// TIA Portal V20 export
FUNCTION "CollectAlarms" : Void   // FC96, LAD
TITLE = Alarm Collector Unit
// Collects alarms from the respective level and categorises the alarms into the different alarm classes.
// stored: Namespace Unit1.Em5, SetENOAutomatically false
   VAR_INPUT
      resetAlarms : Bool;
      disableAlarms : Bool;
   END_VAR
   VAR_OUTPUT
      commandsToUnit : "LUC_typeStateCommands";   // Feedback to the unit
   END_VAR
   VAR CONSTANT
      DelayTime : Time := T#300ms;
      TRUE : Bool := TRUE;
      FALSE : Bool := FALSE;
   END_VAR
BEGIN

REGION Network 1: Reset Alarms
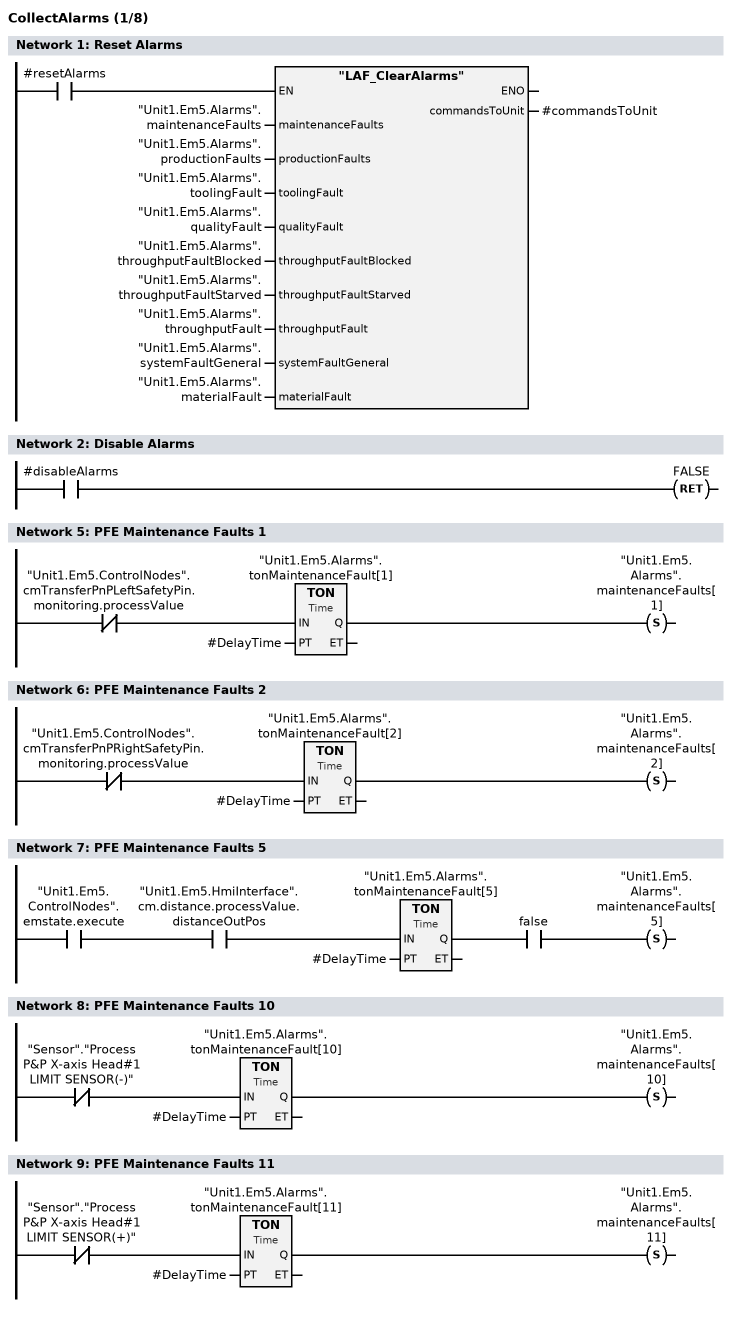
   RUNG wire#powerrail
      Contact( #resetAlarms )
      "LAF_ClearAlarms"(maintenanceFaults := "Unit1.Em5.Alarms".maintenanceFaults, productionFaults := "Unit1.Em5.Alarms".productionFaults, toolingFault := "Unit1.Em5.Alarms".toolingFault, qualityFault := "Unit1.Em5.Alarms".qualityFault, throughputFaultBlocked := "Unit1.Em5.Alarms".throughputFaultBlocked, throughputFaultStarved := "Unit1.Em5.Alarms".throughputFaultStarved, throughputFault := "Unit1.Em5.Alarms".throughputFault, systemFaultGeneral := "Unit1.Em5.Alarms".systemFaultGeneral, materialFault := "Unit1.Em5.Alarms".materialFault, commandsToUnit => #commandsToUnit)
   END_RUNG
   // the same network as SCL:
   IF #resetAlarms THEN
       "LAF_ClearAlarms"(maintenanceFaults := "Unit1.Em5.Alarms".maintenanceFaults,
                         productionFaults := "Unit1.Em5.Alarms".productionFaults,
                         toolingFault := "Unit1.Em5.Alarms".toolingFault,
                         qualityFault := "Unit1.Em5.Alarms".qualityFault,
                         throughputFaultBlocked := "Unit1.Em5.Alarms".throughputFaultBlocked,
                         throughputFaultStarved := "Unit1.Em5.Alarms".throughputFaultStarved,
                         throughputFault := "Unit1.Em5.Alarms".throughputFault,
                         systemFaultGeneral := "Unit1.Em5.Alarms".systemFaultGeneral,
                         materialFault := "Unit1.Em5.Alarms".materialFault,
                         commandsToUnit => #commandsToUnit);
   END_IF;
END_REGION

REGION Network 2: Disable Alarms
   RUNG wire#powerrail
      Contact( #disableAlarms )
      ReturnCoil( FALSE )
   END_RUNG
   // the same network as SCL:
   IF #disableAlarms THEN
       ENO := FALSE;
       RETURN;
   END_IF;
END_REGION

REGION Network 3: *************** Fault ************************
END_REGION

REGION Network 4: PFE Maintenance Faults 0
END_REGION

REGION Network 5: PFE Maintenance Faults 1
   RUNG wire#powerrail
      I_Contact( "Unit1.Em5.ControlNodes".cmTransferPnPLeftSafetyPin.monitoring.processValue )
      { S7_Templates := "time_type := Time" } "Unit1.Em5.Alarms".tonMaintenanceFault[1].TON(pt := #DelayTime, et =>)
      S_Coil( "Unit1.Em5.Alarms".maintenanceFaults[1] )
   END_RUNG
   // the same network as SCL:
   "Unit1.Em5.Alarms".tonMaintenanceFault[1].TON(IN := NOT "Unit1.Em5.ControlNodes".cmTransferPnPLeftSafetyPin.monitoring.processValue,
                           PT := #DelayTime);
   IF "Unit1.Em5.Alarms".tonMaintenanceFault[1].Q THEN
       "Unit1.Em5.Alarms".maintenanceFaults[1] := TRUE;
   END_IF;
END_REGION

REGION Network 6: PFE Maintenance Faults 2
   RUNG wire#powerrail
      I_Contact( "Unit1.Em5.ControlNodes".cmTransferPnPRightSafetyPin.monitoring.processValue )
      { S7_Templates := "time_type := Time" } "Unit1.Em5.Alarms".tonMaintenanceFault[2].TON(pt := #DelayTime, et =>)
      S_Coil( "Unit1.Em5.Alarms".maintenanceFaults[2] )
   END_RUNG
   // the same network as SCL:
   "Unit1.Em5.Alarms".tonMaintenanceFault[2].TON(IN := NOT "Unit1.Em5.ControlNodes".cmTransferPnPRightSafetyPin.monitoring.processValue,
                           PT := #DelayTime);
   IF "Unit1.Em5.Alarms".tonMaintenanceFault[2].Q THEN
       "Unit1.Em5.Alarms".maintenanceFaults[2] := TRUE;
   END_IF;
END_REGION

REGION Network 7: PFE Maintenance Faults 5
   RUNG wire#powerrail
      Contact( "Unit1.Em5.ControlNodes".emstate.execute )
      Contact( "Unit1.Em5.HmiInterface".cm.distance.processValue.distanceOutPos )
      { S7_Templates := "time_type := Time" } "Unit1.Em5.Alarms".tonMaintenanceFault[5].TON(pt := #DelayTime, et =>)
      Contact( false )
      S_Coil( "Unit1.Em5.Alarms".maintenanceFaults[5] )
   END_RUNG
   // the same network as SCL:
   "Unit1.Em5.Alarms".tonMaintenanceFault[5].TON(IN := "Unit1.Em5.ControlNodes".emstate.execute AND "Unit1.Em5.HmiInterface".cm.distance.processValue.distanceOutPos,
                           PT := #DelayTime);
   IF "Unit1.Em5.Alarms".tonMaintenanceFault[5].Q AND false THEN
       "Unit1.Em5.Alarms".maintenanceFaults[5] := TRUE;
   END_IF;
END_REGION

REGION Network 8: PFE Maintenance Faults 10
   RUNG wire#powerrail
      I_Contact( "Sensor"."Process P&P X-axis Head#1 LIMIT SENSOR(-)" )
      { S7_Templates := "time_type := Time" } "Unit1.Em5.Alarms".tonMaintenanceFault[10].TON(pt := #DelayTime, et =>)
      S_Coil( "Unit1.Em5.Alarms".maintenanceFaults[10] )
   END_RUNG
   // the same network as SCL:
   "Unit1.Em5.Alarms".tonMaintenanceFault[10].TON(IN := NOT "Sensor"."Process P&P X-axis Head#1 LIMIT SENSOR(-)",
                           PT := #DelayTime);
   IF "Unit1.Em5.Alarms".tonMaintenanceFault[10].Q THEN
       "Unit1.Em5.Alarms".maintenanceFaults[10] := TRUE;
   END_IF;
END_REGION

REGION Network 9: PFE Maintenance Faults 11
   RUNG wire#powerrail
      I_Contact( "Sensor"."Process P&P X-axis Head#1 LIMIT SENSOR(+)" )
      { S7_Templates := "time_type := Time" } "Unit1.Em5.Alarms".tonMaintenanceFault[11].TON(pt := #DelayTime, et =>)
      S_Coil( "Unit1.Em5.Alarms".maintenanceFaults[11] )
   END_RUNG
   // the same network as SCL:
   "Unit1.Em5.Alarms".tonMaintenanceFault[11].TON(IN := NOT "Sensor"."Process P&P X-axis Head#1 LIMIT SENSOR(+)",
                           PT := #DelayTime);
   IF "Unit1.Em5.Alarms".tonMaintenanceFault[11].Q THEN
       "Unit1.Em5.Alarms".maintenanceFaults[11] := TRUE;
   END_IF;
END_REGION

REGION Network 10: PFE Maintenance Faults 12
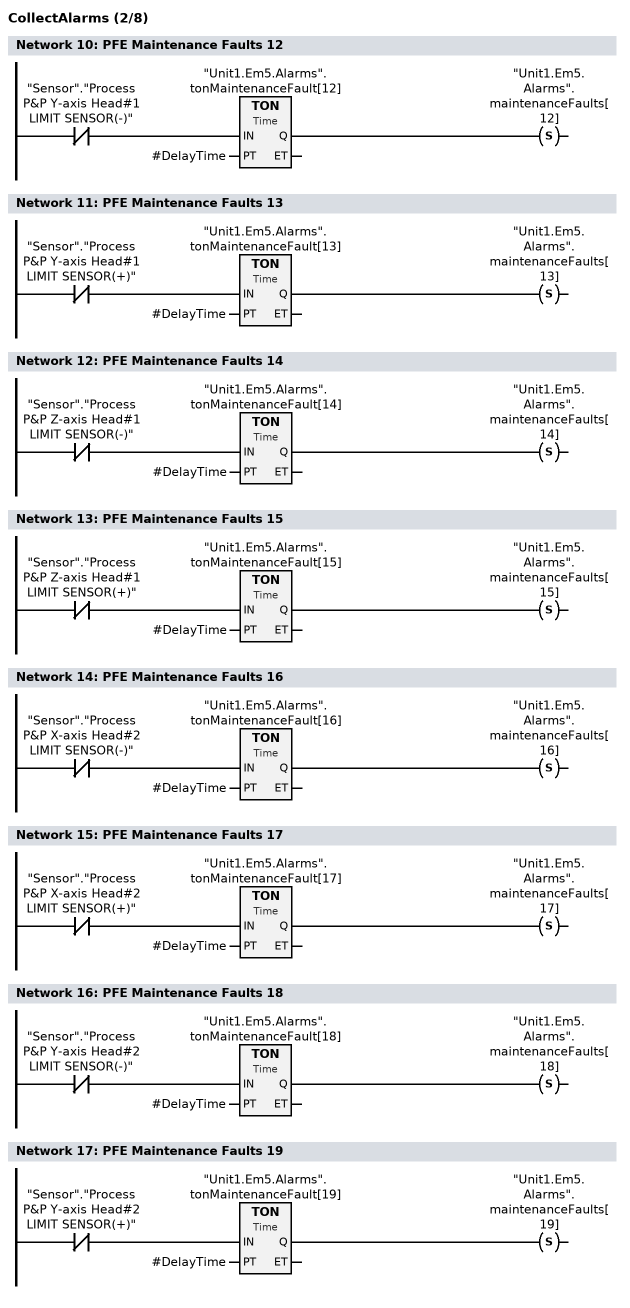
   RUNG wire#powerrail
      I_Contact( "Sensor"."Process P&P Y-axis Head#1 LIMIT SENSOR(-)" )
      { S7_Templates := "time_type := Time" } "Unit1.Em5.Alarms".tonMaintenanceFault[12].TON(pt := #DelayTime, et =>)
      S_Coil( "Unit1.Em5.Alarms".maintenanceFaults[12] )
   END_RUNG
   // the same network as SCL:
   "Unit1.Em5.Alarms".tonMaintenanceFault[12].TON(IN := NOT "Sensor"."Process P&P Y-axis Head#1 LIMIT SENSOR(-)",
                           PT := #DelayTime);
   IF "Unit1.Em5.Alarms".tonMaintenanceFault[12].Q THEN
       "Unit1.Em5.Alarms".maintenanceFaults[12] := TRUE;
   END_IF;
END_REGION

REGION Network 11: PFE Maintenance Faults 13
   RUNG wire#powerrail
      I_Contact( "Sensor"."Process P&P Y-axis Head#1 LIMIT SENSOR(+)" )
      { S7_Templates := "time_type := Time" } "Unit1.Em5.Alarms".tonMaintenanceFault[13].TON(pt := #DelayTime, et =>)
      S_Coil( "Unit1.Em5.Alarms".maintenanceFaults[13] )
   END_RUNG
   // the same network as SCL:
   "Unit1.Em5.Alarms".tonMaintenanceFault[13].TON(IN := NOT "Sensor"."Process P&P Y-axis Head#1 LIMIT SENSOR(+)",
                           PT := #DelayTime);
   IF "Unit1.Em5.Alarms".tonMaintenanceFault[13].Q THEN
       "Unit1.Em5.Alarms".maintenanceFaults[13] := TRUE;
   END_IF;
END_REGION

REGION Network 12: PFE Maintenance Faults 14
   RUNG wire#powerrail
      I_Contact( "Sensor"."Process P&P Z-axis Head#1 LIMIT SENSOR(-)" )
      { S7_Templates := "time_type := Time" } "Unit1.Em5.Alarms".tonMaintenanceFault[14].TON(pt := #DelayTime, et =>)
      S_Coil( "Unit1.Em5.Alarms".maintenanceFaults[14] )
   END_RUNG
   // the same network as SCL:
   "Unit1.Em5.Alarms".tonMaintenanceFault[14].TON(IN := NOT "Sensor"."Process P&P Z-axis Head#1 LIMIT SENSOR(-)",
                           PT := #DelayTime);
   IF "Unit1.Em5.Alarms".tonMaintenanceFault[14].Q THEN
       "Unit1.Em5.Alarms".maintenanceFaults[14] := TRUE;
   END_IF;
END_REGION

REGION Network 13: PFE Maintenance Faults 15
   RUNG wire#powerrail
      I_Contact( "Sensor"."Process P&P Z-axis Head#1 LIMIT SENSOR(+)" )
      { S7_Templates := "time_type := Time" } "Unit1.Em5.Alarms".tonMaintenanceFault[15].TON(pt := #DelayTime, et =>)
      S_Coil( "Unit1.Em5.Alarms".maintenanceFaults[15] )
   END_RUNG
   // the same network as SCL:
   "Unit1.Em5.Alarms".tonMaintenanceFault[15].TON(IN := NOT "Sensor"."Process P&P Z-axis Head#1 LIMIT SENSOR(+)",
                           PT := #DelayTime);
   IF "Unit1.Em5.Alarms".tonMaintenanceFault[15].Q THEN
       "Unit1.Em5.Alarms".maintenanceFaults[15] := TRUE;
   END_IF;
END_REGION

REGION Network 14: PFE Maintenance Faults 16
   RUNG wire#powerrail
      I_Contact( "Sensor"."Process P&P X-axis Head#2 LIMIT SENSOR(-)" )
      { S7_Templates := "time_type := Time" } "Unit1.Em5.Alarms".tonMaintenanceFault[16].TON(pt := #DelayTime, et =>)
      S_Coil( "Unit1.Em5.Alarms".maintenanceFaults[16] )
   END_RUNG
   // the same network as SCL:
   "Unit1.Em5.Alarms".tonMaintenanceFault[16].TON(IN := NOT "Sensor"."Process P&P X-axis Head#2 LIMIT SENSOR(-)",
                           PT := #DelayTime);
   IF "Unit1.Em5.Alarms".tonMaintenanceFault[16].Q THEN
       "Unit1.Em5.Alarms".maintenanceFaults[16] := TRUE;
   END_IF;
END_REGION

REGION Network 15: PFE Maintenance Faults 17
   RUNG wire#powerrail
      I_Contact( "Sensor"."Process P&P X-axis Head#2 LIMIT SENSOR(+)" )
      { S7_Templates := "time_type := Time" } "Unit1.Em5.Alarms".tonMaintenanceFault[17].TON(pt := #DelayTime, et =>)
      S_Coil( "Unit1.Em5.Alarms".maintenanceFaults[17] )
   END_RUNG
   // the same network as SCL:
   "Unit1.Em5.Alarms".tonMaintenanceFault[17].TON(IN := NOT "Sensor"."Process P&P X-axis Head#2 LIMIT SENSOR(+)",
                           PT := #DelayTime);
   IF "Unit1.Em5.Alarms".tonMaintenanceFault[17].Q THEN
       "Unit1.Em5.Alarms".maintenanceFaults[17] := TRUE;
   END_IF;
END_REGION

REGION Network 16: PFE Maintenance Faults 18
   RUNG wire#powerrail
      I_Contact( "Sensor"."Process P&P Y-axis Head#2 LIMIT SENSOR(-)" )
      { S7_Templates := "time_type := Time" } "Unit1.Em5.Alarms".tonMaintenanceFault[18].TON(pt := #DelayTime, et =>)
      S_Coil( "Unit1.Em5.Alarms".maintenanceFaults[18] )
   END_RUNG
   // the same network as SCL:
   "Unit1.Em5.Alarms".tonMaintenanceFault[18].TON(IN := NOT "Sensor"."Process P&P Y-axis Head#2 LIMIT SENSOR(-)",
                           PT := #DelayTime);
   IF "Unit1.Em5.Alarms".tonMaintenanceFault[18].Q THEN
       "Unit1.Em5.Alarms".maintenanceFaults[18] := TRUE;
   END_IF;
END_REGION

REGION Network 17: PFE Maintenance Faults 19
   RUNG wire#powerrail
      I_Contact( "Sensor"."Process P&P Y-axis Head#2 LIMIT SENSOR(+)" )
      { S7_Templates := "time_type := Time" } "Unit1.Em5.Alarms".tonMaintenanceFault[19].TON(pt := #DelayTime, et =>)
      S_Coil( "Unit1.Em5.Alarms".maintenanceFaults[19] )
   END_RUNG
   // the same network as SCL:
   "Unit1.Em5.Alarms".tonMaintenanceFault[19].TON(IN := NOT "Sensor"."Process P&P Y-axis Head#2 LIMIT SENSOR(+)",
                           PT := #DelayTime);
   IF "Unit1.Em5.Alarms".tonMaintenanceFault[19].Q THEN
       "Unit1.Em5.Alarms".maintenanceFaults[19] := TRUE;
   END_IF;
END_REGION

REGION Network 18: PFE Maintenance Faults 20
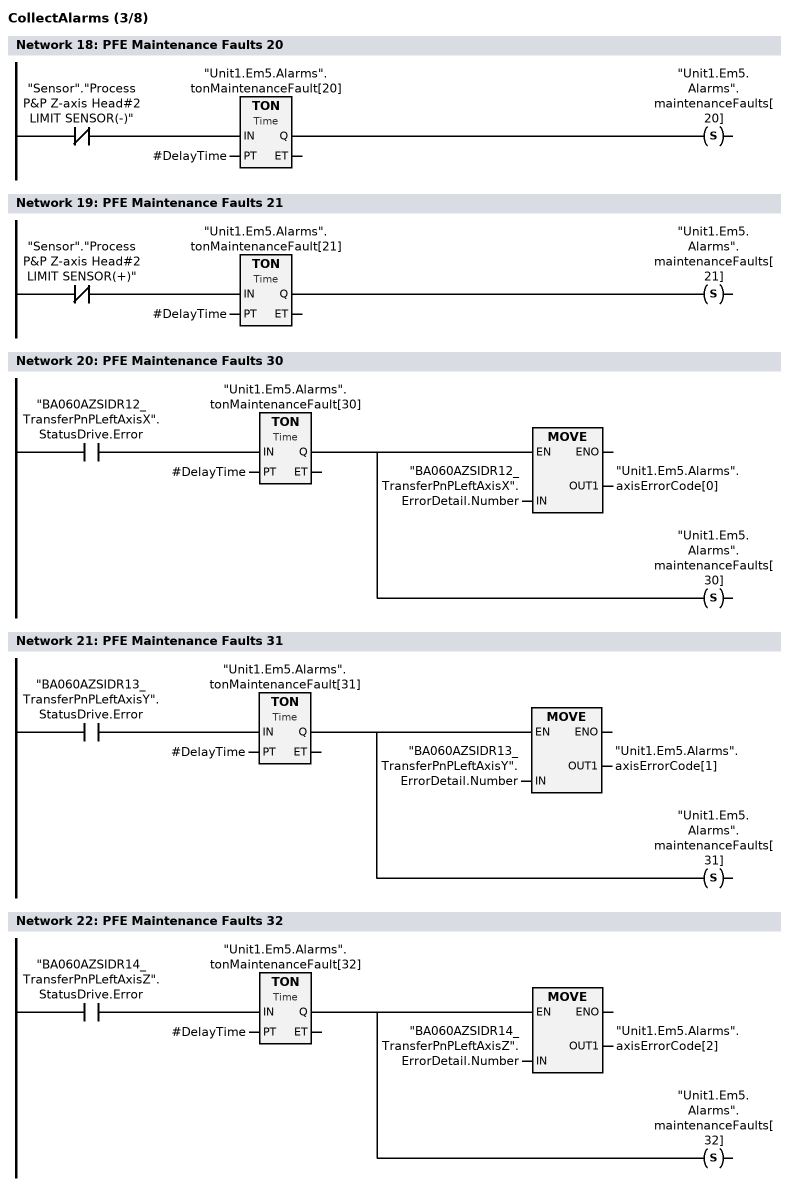
   RUNG wire#powerrail
      I_Contact( "Sensor"."Process P&P Z-axis Head#2 LIMIT SENSOR(-)" )
      { S7_Templates := "time_type := Time" } "Unit1.Em5.Alarms".tonMaintenanceFault[20].TON(pt := #DelayTime, et =>)
      S_Coil( "Unit1.Em5.Alarms".maintenanceFaults[20] )
   END_RUNG
   // the same network as SCL:
   "Unit1.Em5.Alarms".tonMaintenanceFault[20].TON(IN := NOT "Sensor"."Process P&P Z-axis Head#2 LIMIT SENSOR(-)",
                           PT := #DelayTime);
   IF "Unit1.Em5.Alarms".tonMaintenanceFault[20].Q THEN
       "Unit1.Em5.Alarms".maintenanceFaults[20] := TRUE;
   END_IF;
END_REGION

REGION Network 19: PFE Maintenance Faults 21
   RUNG wire#powerrail
      I_Contact( "Sensor"."Process P&P Z-axis Head#2 LIMIT SENSOR(+)" )
      { S7_Templates := "time_type := Time" } "Unit1.Em5.Alarms".tonMaintenanceFault[21].TON(pt := #DelayTime, et =>)
      S_Coil( "Unit1.Em5.Alarms".maintenanceFaults[21] )
   END_RUNG
   // the same network as SCL:
   "Unit1.Em5.Alarms".tonMaintenanceFault[21].TON(IN := NOT "Sensor"."Process P&P Z-axis Head#2 LIMIT SENSOR(+)",
                           PT := #DelayTime);
   IF "Unit1.Em5.Alarms".tonMaintenanceFault[21].Q THEN
       "Unit1.Em5.Alarms".maintenanceFaults[21] := TRUE;
   END_IF;
END_REGION

REGION Network 20: PFE Maintenance Faults 30
   RUNG wire#powerrail
      Contact( "BA060AZSIDR12_TransferPnPLeftAxisX".StatusDrive.Error )
      { S7_Templates := "time_type := Time" } "Unit1.Em5.Alarms".tonMaintenanceFault[30].TON(pt := #DelayTime, et =>)
      wire#w1
      Move(in := "BA060AZSIDR12_TransferPnPLeftAxisX".ErrorDetail.Number, out1 => "Unit1.Em5.Alarms".axisErrorCode[0])
   END_RUNG
   RUNG wire#w1
      S_Coil( "Unit1.Em5.Alarms".maintenanceFaults[30] )
   END_RUNG
   // the same network as SCL:
   "Unit1.Em5.Alarms".tonMaintenanceFault[30].TON(IN := "BA060AZSIDR12_TransferPnPLeftAxisX".StatusDrive.Error,
                           PT := #DelayTime);
   IF "Unit1.Em5.Alarms".tonMaintenanceFault[30].Q THEN
       "Unit1.Em5.Alarms".axisErrorCode[0] := "BA060AZSIDR12_TransferPnPLeftAxisX".ErrorDetail.Number;
       "Unit1.Em5.Alarms".maintenanceFaults[30] := TRUE;
   END_IF;
END_REGION

REGION Network 21: PFE Maintenance Faults 31
   RUNG wire#powerrail
      Contact( "BA060AZSIDR13_TransferPnPLeftAxisY".StatusDrive.Error )
      { S7_Templates := "time_type := Time" } "Unit1.Em5.Alarms".tonMaintenanceFault[31].TON(pt := #DelayTime, et =>)
      wire#w1
      Move(in := "BA060AZSIDR13_TransferPnPLeftAxisY".ErrorDetail.Number, out1 => "Unit1.Em5.Alarms".axisErrorCode[1])
   END_RUNG
   RUNG wire#w1
      S_Coil( "Unit1.Em5.Alarms".maintenanceFaults[31] )
   END_RUNG
   // the same network as SCL:
   "Unit1.Em5.Alarms".tonMaintenanceFault[31].TON(IN := "BA060AZSIDR13_TransferPnPLeftAxisY".StatusDrive.Error,
                           PT := #DelayTime);
   IF "Unit1.Em5.Alarms".tonMaintenanceFault[31].Q THEN
       "Unit1.Em5.Alarms".axisErrorCode[1] := "BA060AZSIDR13_TransferPnPLeftAxisY".ErrorDetail.Number;
       "Unit1.Em5.Alarms".maintenanceFaults[31] := TRUE;
   END_IF;
END_REGION

REGION Network 22: PFE Maintenance Faults 32
   RUNG wire#powerrail
      Contact( "BA060AZSIDR14_TransferPnPLeftAxisZ".StatusDrive.Error )
      { S7_Templates := "time_type := Time" } "Unit1.Em5.Alarms".tonMaintenanceFault[32].TON(pt := #DelayTime, et =>)
      wire#w1
      Move(in := "BA060AZSIDR14_TransferPnPLeftAxisZ".ErrorDetail.Number, out1 => "Unit1.Em5.Alarms".axisErrorCode[2])
   END_RUNG
   RUNG wire#w1
      S_Coil( "Unit1.Em5.Alarms".maintenanceFaults[32] )
   END_RUNG
   // the same network as SCL:
   "Unit1.Em5.Alarms".tonMaintenanceFault[32].TON(IN := "BA060AZSIDR14_TransferPnPLeftAxisZ".StatusDrive.Error,
                           PT := #DelayTime);
   IF "Unit1.Em5.Alarms".tonMaintenanceFault[32].Q THEN
       "Unit1.Em5.Alarms".axisErrorCode[2] := "BA060AZSIDR14_TransferPnPLeftAxisZ".ErrorDetail.Number;
       "Unit1.Em5.Alarms".maintenanceFaults[32] := TRUE;
   END_IF;
END_REGION

REGION Network 23: PFE Maintenance Faults 33
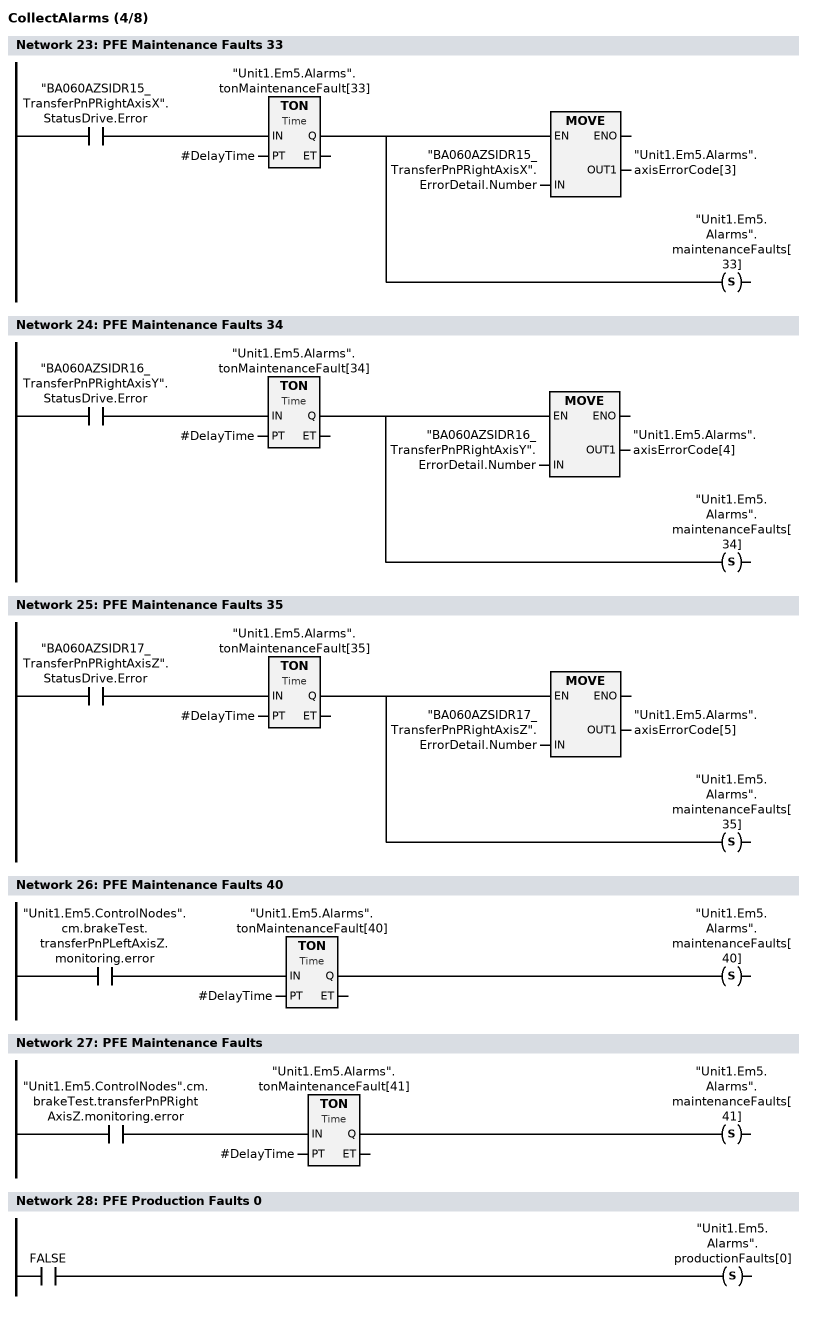
   RUNG wire#powerrail
      Contact( "BA060AZSIDR15_TransferPnPRightAxisX".StatusDrive.Error )
      { S7_Templates := "time_type := Time" } "Unit1.Em5.Alarms".tonMaintenanceFault[33].TON(pt := #DelayTime, et =>)
      wire#w1
      Move(in := "BA060AZSIDR15_TransferPnPRightAxisX".ErrorDetail.Number, out1 => "Unit1.Em5.Alarms".axisErrorCode[3])
   END_RUNG
   RUNG wire#w1
      S_Coil( "Unit1.Em5.Alarms".maintenanceFaults[33] )
   END_RUNG
   // the same network as SCL:
   "Unit1.Em5.Alarms".tonMaintenanceFault[33].TON(IN := "BA060AZSIDR15_TransferPnPRightAxisX".StatusDrive.Error,
                           PT := #DelayTime);
   IF "Unit1.Em5.Alarms".tonMaintenanceFault[33].Q THEN
       "Unit1.Em5.Alarms".axisErrorCode[3] := "BA060AZSIDR15_TransferPnPRightAxisX".ErrorDetail.Number;
       "Unit1.Em5.Alarms".maintenanceFaults[33] := TRUE;
   END_IF;
END_REGION

REGION Network 24: PFE Maintenance Faults 34
   RUNG wire#powerrail
      Contact( "BA060AZSIDR16_TransferPnPRightAxisY".StatusDrive.Error )
      { S7_Templates := "time_type := Time" } "Unit1.Em5.Alarms".tonMaintenanceFault[34].TON(pt := #DelayTime, et =>)
      wire#w1
      Move(in := "BA060AZSIDR16_TransferPnPRightAxisY".ErrorDetail.Number, out1 => "Unit1.Em5.Alarms".axisErrorCode[4])
   END_RUNG
   RUNG wire#w1
      S_Coil( "Unit1.Em5.Alarms".maintenanceFaults[34] )
   END_RUNG
   // the same network as SCL:
   "Unit1.Em5.Alarms".tonMaintenanceFault[34].TON(IN := "BA060AZSIDR16_TransferPnPRightAxisY".StatusDrive.Error,
                           PT := #DelayTime);
   IF "Unit1.Em5.Alarms".tonMaintenanceFault[34].Q THEN
       "Unit1.Em5.Alarms".axisErrorCode[4] := "BA060AZSIDR16_TransferPnPRightAxisY".ErrorDetail.Number;
       "Unit1.Em5.Alarms".maintenanceFaults[34] := TRUE;
   END_IF;
END_REGION

REGION Network 25: PFE Maintenance Faults 35
   RUNG wire#powerrail
      Contact( "BA060AZSIDR17_TransferPnPRightAxisZ".StatusDrive.Error )
      { S7_Templates := "time_type := Time" } "Unit1.Em5.Alarms".tonMaintenanceFault[35].TON(pt := #DelayTime, et =>)
      wire#w1
      Move(in := "BA060AZSIDR17_TransferPnPRightAxisZ".ErrorDetail.Number, out1 => "Unit1.Em5.Alarms".axisErrorCode[5])
   END_RUNG
   RUNG wire#w1
      S_Coil( "Unit1.Em5.Alarms".maintenanceFaults[35] )
   END_RUNG
   // the same network as SCL:
   "Unit1.Em5.Alarms".tonMaintenanceFault[35].TON(IN := "BA060AZSIDR17_TransferPnPRightAxisZ".StatusDrive.Error,
                           PT := #DelayTime);
   IF "Unit1.Em5.Alarms".tonMaintenanceFault[35].Q THEN
       "Unit1.Em5.Alarms".axisErrorCode[5] := "BA060AZSIDR17_TransferPnPRightAxisZ".ErrorDetail.Number;
       "Unit1.Em5.Alarms".maintenanceFaults[35] := TRUE;
   END_IF;
END_REGION

REGION Network 26: PFE Maintenance Faults 40
   RUNG wire#powerrail
      Contact( "Unit1.Em5.ControlNodes".cm.brakeTest.transferPnPLeftAxisZ.monitoring.error )
      { S7_Templates := "time_type := Time" } "Unit1.Em5.Alarms".tonMaintenanceFault[40].TON(pt := #DelayTime, et =>)
      S_Coil( "Unit1.Em5.Alarms".maintenanceFaults[40] )
   END_RUNG
   // the same network as SCL:
   "Unit1.Em5.Alarms".tonMaintenanceFault[40].TON(IN := "Unit1.Em5.ControlNodes".cm.brakeTest.transferPnPLeftAxisZ.monitoring.error,
                           PT := #DelayTime);
   IF "Unit1.Em5.Alarms".tonMaintenanceFault[40].Q THEN
       "Unit1.Em5.Alarms".maintenanceFaults[40] := TRUE;
   END_IF;
END_REGION

REGION Network 27: PFE Maintenance Faults
   RUNG wire#powerrail
      Contact( "Unit1.Em5.ControlNodes".cm.brakeTest.transferPnPRightAxisZ.monitoring.error )
      { S7_Templates := "time_type := Time" } "Unit1.Em5.Alarms".tonMaintenanceFault[41].TON(pt := #DelayTime, et =>)
      S_Coil( "Unit1.Em5.Alarms".maintenanceFaults[41] )
   END_RUNG
   // the same network as SCL:
   "Unit1.Em5.Alarms".tonMaintenanceFault[41].TON(IN := "Unit1.Em5.ControlNodes".cm.brakeTest.transferPnPRightAxisZ.monitoring.error,
                           PT := #DelayTime);
   IF "Unit1.Em5.Alarms".tonMaintenanceFault[41].Q THEN
       "Unit1.Em5.Alarms".maintenanceFaults[41] := TRUE;
   END_IF;
END_REGION

REGION Network 28: PFE Production Faults 0
   RUNG wire#powerrail
      Contact( FALSE )
      S_Coil( "Unit1.Em5.Alarms".productionFaults[0] )
   END_RUNG
   // the same network as SCL:
   IF FALSE THEN "Unit1.Em5.Alarms".productionFaults[0] := TRUE; END_IF;
END_REGION

REGION Network 29: PFE Production Faults 1
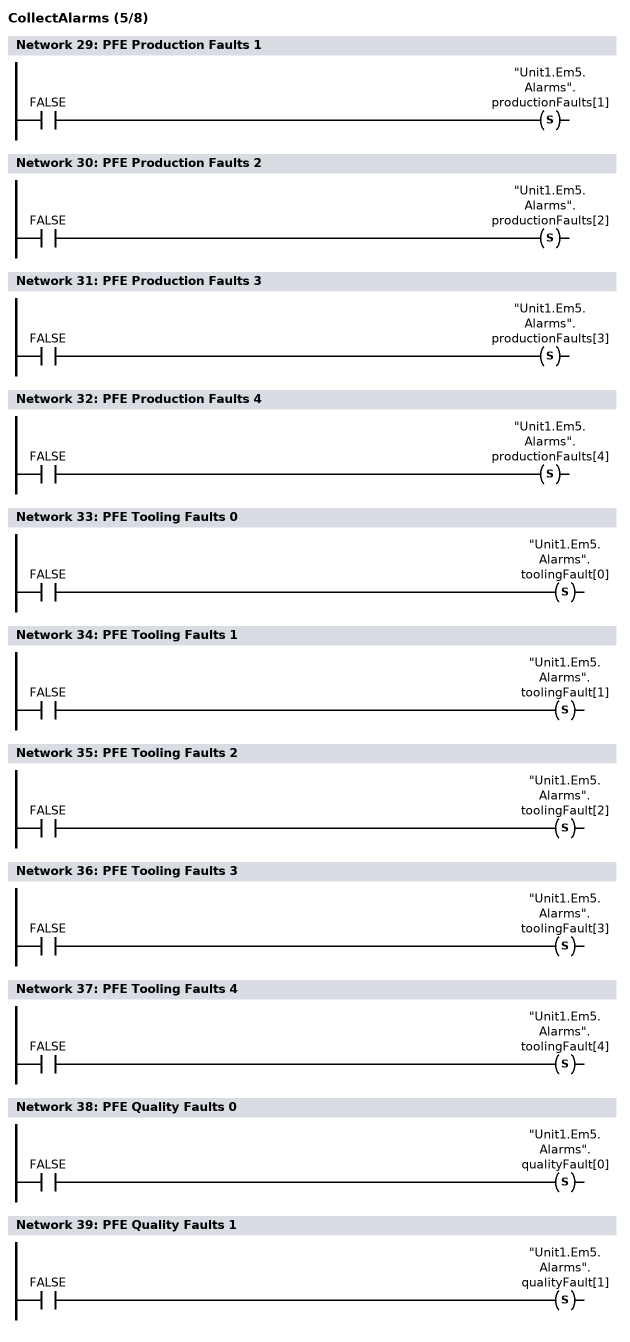
   RUNG wire#powerrail
      Contact( FALSE )
      S_Coil( "Unit1.Em5.Alarms".productionFaults[1] )
   END_RUNG
   // the same network as SCL:
   IF FALSE THEN "Unit1.Em5.Alarms".productionFaults[1] := TRUE; END_IF;
END_REGION

REGION Network 30: PFE Production Faults 2
   RUNG wire#powerrail
      Contact( FALSE )
      S_Coil( "Unit1.Em5.Alarms".productionFaults[2] )
   END_RUNG
   // the same network as SCL:
   IF FALSE THEN "Unit1.Em5.Alarms".productionFaults[2] := TRUE; END_IF;
END_REGION

REGION Network 31: PFE Production Faults 3
   RUNG wire#powerrail
      Contact( FALSE )
      S_Coil( "Unit1.Em5.Alarms".productionFaults[3] )
   END_RUNG
   // the same network as SCL:
   IF FALSE THEN "Unit1.Em5.Alarms".productionFaults[3] := TRUE; END_IF;
END_REGION

REGION Network 32: PFE Production Faults 4
   RUNG wire#powerrail
      Contact( FALSE )
      S_Coil( "Unit1.Em5.Alarms".productionFaults[4] )
   END_RUNG
   // the same network as SCL:
   IF FALSE THEN "Unit1.Em5.Alarms".productionFaults[4] := TRUE; END_IF;
END_REGION

REGION Network 33: PFE Tooling Faults 0
   RUNG wire#powerrail
      Contact( FALSE )
      S_Coil( "Unit1.Em5.Alarms".toolingFault[0] )
   END_RUNG
   // the same network as SCL:
   IF FALSE THEN "Unit1.Em5.Alarms".toolingFault[0] := TRUE; END_IF;
END_REGION

REGION Network 34: PFE Tooling Faults 1
   RUNG wire#powerrail
      Contact( FALSE )
      S_Coil( "Unit1.Em5.Alarms".toolingFault[1] )
   END_RUNG
   // the same network as SCL:
   IF FALSE THEN "Unit1.Em5.Alarms".toolingFault[1] := TRUE; END_IF;
END_REGION

REGION Network 35: PFE Tooling Faults 2
   RUNG wire#powerrail
      Contact( FALSE )
      S_Coil( "Unit1.Em5.Alarms".toolingFault[2] )
   END_RUNG
   // the same network as SCL:
   IF FALSE THEN "Unit1.Em5.Alarms".toolingFault[2] := TRUE; END_IF;
END_REGION

REGION Network 36: PFE Tooling Faults 3
   RUNG wire#powerrail
      Contact( FALSE )
      S_Coil( "Unit1.Em5.Alarms".toolingFault[3] )
   END_RUNG
   // the same network as SCL:
   IF FALSE THEN "Unit1.Em5.Alarms".toolingFault[3] := TRUE; END_IF;
END_REGION

REGION Network 37: PFE Tooling Faults 4
   RUNG wire#powerrail
      Contact( FALSE )
      S_Coil( "Unit1.Em5.Alarms".toolingFault[4] )
   END_RUNG
   // the same network as SCL:
   IF FALSE THEN "Unit1.Em5.Alarms".toolingFault[4] := TRUE; END_IF;
END_REGION

REGION Network 38: PFE Quality Faults 0
   RUNG wire#powerrail
      Contact( FALSE )
      S_Coil( "Unit1.Em5.Alarms".qualityFault[0] )
   END_RUNG
   // the same network as SCL:
   IF FALSE THEN "Unit1.Em5.Alarms".qualityFault[0] := TRUE; END_IF;
END_REGION

REGION Network 39: PFE Quality Faults 1
   RUNG wire#powerrail
      Contact( FALSE )
      S_Coil( "Unit1.Em5.Alarms".qualityFault[1] )
   END_RUNG
   // the same network as SCL:
   IF FALSE THEN "Unit1.Em5.Alarms".qualityFault[1] := TRUE; END_IF;
END_REGION

REGION Network 40: PFE Quality Faults 2
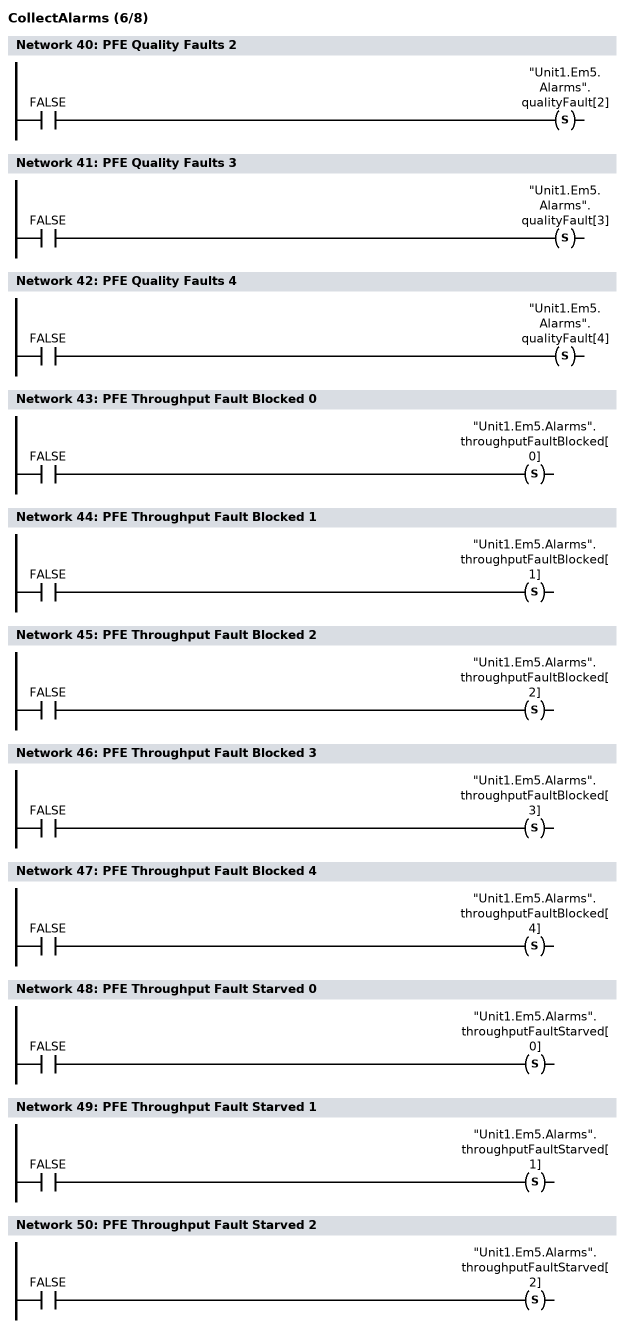
   RUNG wire#powerrail
      Contact( FALSE )
      S_Coil( "Unit1.Em5.Alarms".qualityFault[2] )
   END_RUNG
   // the same network as SCL:
   IF FALSE THEN "Unit1.Em5.Alarms".qualityFault[2] := TRUE; END_IF;
END_REGION

REGION Network 41: PFE Quality Faults 3
   RUNG wire#powerrail
      Contact( FALSE )
      S_Coil( "Unit1.Em5.Alarms".qualityFault[3] )
   END_RUNG
   // the same network as SCL:
   IF FALSE THEN "Unit1.Em5.Alarms".qualityFault[3] := TRUE; END_IF;
END_REGION

REGION Network 42: PFE Quality Faults 4
   RUNG wire#powerrail
      Contact( FALSE )
      S_Coil( "Unit1.Em5.Alarms".qualityFault[4] )
   END_RUNG
   // the same network as SCL:
   IF FALSE THEN "Unit1.Em5.Alarms".qualityFault[4] := TRUE; END_IF;
END_REGION

REGION Network 43: PFE Throughput Fault Blocked 0
   RUNG wire#powerrail
      Contact( FALSE )
      S_Coil( "Unit1.Em5.Alarms".throughputFaultBlocked[0] )
   END_RUNG
   // the same network as SCL:
   IF FALSE THEN "Unit1.Em5.Alarms".throughputFaultBlocked[0] := TRUE; END_IF;
END_REGION

REGION Network 44: PFE Throughput Fault Blocked 1
   RUNG wire#powerrail
      Contact( FALSE )
      S_Coil( "Unit1.Em5.Alarms".throughputFaultBlocked[1] )
   END_RUNG
   // the same network as SCL:
   IF FALSE THEN "Unit1.Em5.Alarms".throughputFaultBlocked[1] := TRUE; END_IF;
END_REGION

REGION Network 45: PFE Throughput Fault Blocked 2
   RUNG wire#powerrail
      Contact( FALSE )
      S_Coil( "Unit1.Em5.Alarms".throughputFaultBlocked[2] )
   END_RUNG
   // the same network as SCL:
   IF FALSE THEN "Unit1.Em5.Alarms".throughputFaultBlocked[2] := TRUE; END_IF;
END_REGION

REGION Network 46: PFE Throughput Fault Blocked 3
   RUNG wire#powerrail
      Contact( FALSE )
      S_Coil( "Unit1.Em5.Alarms".throughputFaultBlocked[3] )
   END_RUNG
   // the same network as SCL:
   IF FALSE THEN "Unit1.Em5.Alarms".throughputFaultBlocked[3] := TRUE; END_IF;
END_REGION

REGION Network 47: PFE Throughput Fault Blocked 4
   RUNG wire#powerrail
      Contact( FALSE )
      S_Coil( "Unit1.Em5.Alarms".throughputFaultBlocked[4] )
   END_RUNG
   // the same network as SCL:
   IF FALSE THEN "Unit1.Em5.Alarms".throughputFaultBlocked[4] := TRUE; END_IF;
END_REGION

REGION Network 48: PFE Throughput Fault Starved 0
   RUNG wire#powerrail
      Contact( FALSE )
      S_Coil( "Unit1.Em5.Alarms".throughputFaultStarved[0] )
   END_RUNG
   // the same network as SCL:
   IF FALSE THEN "Unit1.Em5.Alarms".throughputFaultStarved[0] := TRUE; END_IF;
END_REGION

REGION Network 49: PFE Throughput Fault Starved 1
   RUNG wire#powerrail
      Contact( FALSE )
      S_Coil( "Unit1.Em5.Alarms".throughputFaultStarved[1] )
   END_RUNG
   // the same network as SCL:
   IF FALSE THEN "Unit1.Em5.Alarms".throughputFaultStarved[1] := TRUE; END_IF;
END_REGION

REGION Network 50: PFE Throughput Fault Starved 2
   RUNG wire#powerrail
      Contact( FALSE )
      S_Coil( "Unit1.Em5.Alarms".throughputFaultStarved[2] )
   END_RUNG
   // the same network as SCL:
   IF FALSE THEN "Unit1.Em5.Alarms".throughputFaultStarved[2] := TRUE; END_IF;
END_REGION

REGION Network 51: PFE Throughput Fault Starved 3
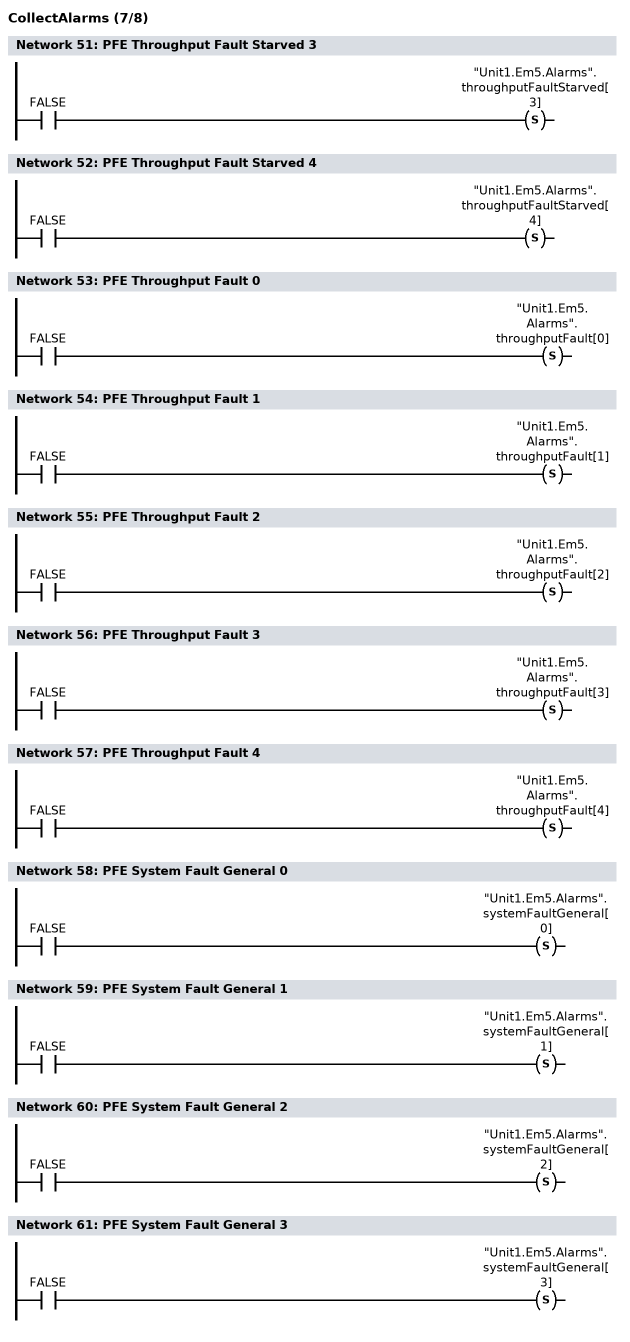
   RUNG wire#powerrail
      Contact( FALSE )
      S_Coil( "Unit1.Em5.Alarms".throughputFaultStarved[3] )
   END_RUNG
   // the same network as SCL:
   IF FALSE THEN "Unit1.Em5.Alarms".throughputFaultStarved[3] := TRUE; END_IF;
END_REGION

REGION Network 52: PFE Throughput Fault Starved 4
   RUNG wire#powerrail
      Contact( FALSE )
      S_Coil( "Unit1.Em5.Alarms".throughputFaultStarved[4] )
   END_RUNG
   // the same network as SCL:
   IF FALSE THEN "Unit1.Em5.Alarms".throughputFaultStarved[4] := TRUE; END_IF;
END_REGION

REGION Network 53: PFE Throughput Fault 0
   RUNG wire#powerrail
      Contact( FALSE )
      S_Coil( "Unit1.Em5.Alarms".throughputFault[0] )
   END_RUNG
   // the same network as SCL:
   IF FALSE THEN "Unit1.Em5.Alarms".throughputFault[0] := TRUE; END_IF;
END_REGION

REGION Network 54: PFE Throughput Fault 1
   RUNG wire#powerrail
      Contact( FALSE )
      S_Coil( "Unit1.Em5.Alarms".throughputFault[1] )
   END_RUNG
   // the same network as SCL:
   IF FALSE THEN "Unit1.Em5.Alarms".throughputFault[1] := TRUE; END_IF;
END_REGION

REGION Network 55: PFE Throughput Fault 2
   RUNG wire#powerrail
      Contact( FALSE )
      S_Coil( "Unit1.Em5.Alarms".throughputFault[2] )
   END_RUNG
   // the same network as SCL:
   IF FALSE THEN "Unit1.Em5.Alarms".throughputFault[2] := TRUE; END_IF;
END_REGION

REGION Network 56: PFE Throughput Fault 3
   RUNG wire#powerrail
      Contact( FALSE )
      S_Coil( "Unit1.Em5.Alarms".throughputFault[3] )
   END_RUNG
   // the same network as SCL:
   IF FALSE THEN "Unit1.Em5.Alarms".throughputFault[3] := TRUE; END_IF;
END_REGION

REGION Network 57: PFE Throughput Fault 4
   RUNG wire#powerrail
      Contact( FALSE )
      S_Coil( "Unit1.Em5.Alarms".throughputFault[4] )
   END_RUNG
   // the same network as SCL:
   IF FALSE THEN "Unit1.Em5.Alarms".throughputFault[4] := TRUE; END_IF;
END_REGION

REGION Network 58: PFE System Fault General 0
   RUNG wire#powerrail
      Contact( FALSE )
      S_Coil( "Unit1.Em5.Alarms".systemFaultGeneral[0] )
   END_RUNG
   // the same network as SCL:
   IF FALSE THEN "Unit1.Em5.Alarms".systemFaultGeneral[0] := TRUE; END_IF;
END_REGION

REGION Network 59: PFE System Fault General 1
   RUNG wire#powerrail
      Contact( FALSE )
      S_Coil( "Unit1.Em5.Alarms".systemFaultGeneral[1] )
   END_RUNG
   // the same network as SCL:
   IF FALSE THEN "Unit1.Em5.Alarms".systemFaultGeneral[1] := TRUE; END_IF;
END_REGION

REGION Network 60: PFE System Fault General 2
   RUNG wire#powerrail
      Contact( FALSE )
      S_Coil( "Unit1.Em5.Alarms".systemFaultGeneral[2] )
   END_RUNG
   // the same network as SCL:
   IF FALSE THEN "Unit1.Em5.Alarms".systemFaultGeneral[2] := TRUE; END_IF;
END_REGION

REGION Network 61: PFE System Fault General 3
   RUNG wire#powerrail
      Contact( FALSE )
      S_Coil( "Unit1.Em5.Alarms".systemFaultGeneral[3] )
   END_RUNG
   // the same network as SCL:
   IF FALSE THEN "Unit1.Em5.Alarms".systemFaultGeneral[3] := TRUE; END_IF;
END_REGION

REGION Network 62: PFE System Fault General 4
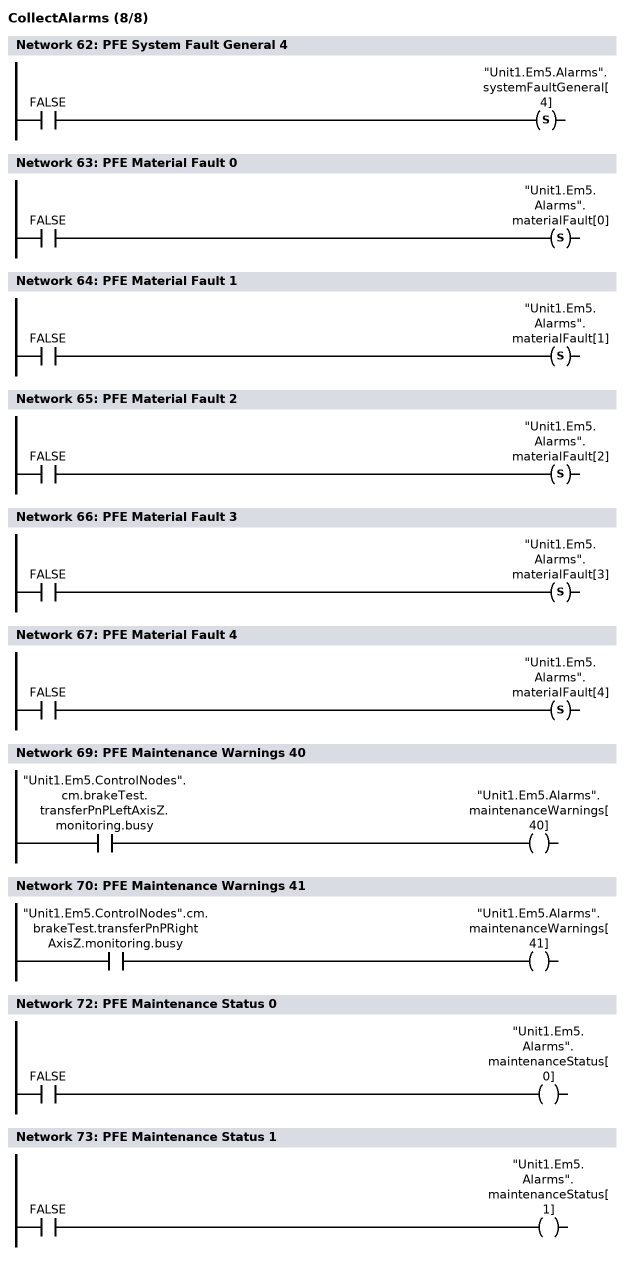
   RUNG wire#powerrail
      Contact( FALSE )
      S_Coil( "Unit1.Em5.Alarms".systemFaultGeneral[4] )
   END_RUNG
   // the same network as SCL:
   IF FALSE THEN "Unit1.Em5.Alarms".systemFaultGeneral[4] := TRUE; END_IF;
END_REGION

REGION Network 63: PFE Material Fault 0
   RUNG wire#powerrail
      Contact( FALSE )
      S_Coil( "Unit1.Em5.Alarms".materialFault[0] )
   END_RUNG
   // the same network as SCL:
   IF FALSE THEN "Unit1.Em5.Alarms".materialFault[0] := TRUE; END_IF;
END_REGION

REGION Network 64: PFE Material Fault 1
   RUNG wire#powerrail
      Contact( FALSE )
      S_Coil( "Unit1.Em5.Alarms".materialFault[1] )
   END_RUNG
   // the same network as SCL:
   IF FALSE THEN "Unit1.Em5.Alarms".materialFault[1] := TRUE; END_IF;
END_REGION

REGION Network 65: PFE Material Fault 2
   RUNG wire#powerrail
      Contact( FALSE )
      S_Coil( "Unit1.Em5.Alarms".materialFault[2] )
   END_RUNG
   // the same network as SCL:
   IF FALSE THEN "Unit1.Em5.Alarms".materialFault[2] := TRUE; END_IF;
END_REGION

REGION Network 66: PFE Material Fault 3
   RUNG wire#powerrail
      Contact( FALSE )
      S_Coil( "Unit1.Em5.Alarms".materialFault[3] )
   END_RUNG
   // the same network as SCL:
   IF FALSE THEN "Unit1.Em5.Alarms".materialFault[3] := TRUE; END_IF;
END_REGION

REGION Network 67: PFE Material Fault 4
   RUNG wire#powerrail
      Contact( FALSE )
      S_Coil( "Unit1.Em5.Alarms".materialFault[4] )
   END_RUNG
   // the same network as SCL:
   IF FALSE THEN "Unit1.Em5.Alarms".materialFault[4] := TRUE; END_IF;
END_REGION

REGION Network 68: ******************** Warning ********************
END_REGION

REGION Network 69: PFE Maintenance Warnings 40
   RUNG wire#powerrail
      Contact( "Unit1.Em5.ControlNodes".cm.brakeTest.transferPnPLeftAxisZ.monitoring.busy )
      Coil( "Unit1.Em5.Alarms".maintenanceWarnings[40] )
   END_RUNG
   // the same network as SCL:
   "Unit1.Em5.Alarms".maintenanceWarnings[40] := "Unit1.Em5.ControlNodes".cm.brakeTest.transferPnPLeftAxisZ.monitoring.busy;
END_REGION

REGION Network 70: PFE Maintenance Warnings 41
   RUNG wire#powerrail
      Contact( "Unit1.Em5.ControlNodes".cm.brakeTest.transferPnPRightAxisZ.monitoring.busy )
      Coil( "Unit1.Em5.Alarms".maintenanceWarnings[41] )
   END_RUNG
   // the same network as SCL:
   "Unit1.Em5.Alarms".maintenanceWarnings[41] := "Unit1.Em5.ControlNodes".cm.brakeTest.transferPnPRightAxisZ.monitoring.busy;
END_REGION

REGION Network 71: ******************** Status ********************
END_REGION

REGION Network 72: PFE Maintenance Status 0
   RUNG wire#powerrail
      Contact( FALSE )
      Coil( "Unit1.Em5.Alarms".maintenanceStatus[0] )
   END_RUNG
   // the same network as SCL:
   "Unit1.Em5.Alarms".maintenanceStatus[0] := FALSE;
END_REGION

REGION Network 73: PFE Maintenance Status 1
   RUNG wire#powerrail
      Contact( FALSE )
      Coil( "Unit1.Em5.Alarms".maintenanceStatus[1] )
   END_RUNG
   // the same network as SCL:
   "Unit1.Em5.Alarms".maintenanceStatus[1] := FALSE;
END_REGION
END_FUNCTION
